// Mitsubishi GX Works2 project: new tz mechanism   PLC: FX3U/FX3UC

PROGRAM MAIN
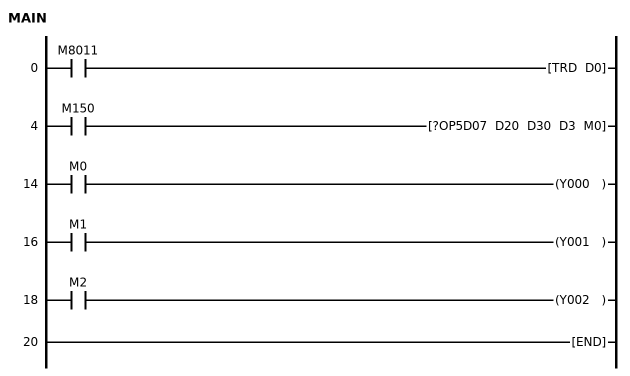
0     LD      M8011
      TRD     D0
4     LD      M150
      ?OP5D07 D20 D30 D3 M0
14    LD      M0
      OUT     Y000
16    LD      M1
      OUT     Y001
18    LD      M2
      OUT     Y002
20    END
END_PROGRAM
